FUNCTION_BLOCK FB_TaskMoveA_tilt EXTENDS FB_AbstructFuture
VAR_OUTPUT
END_VAR
VAR
	_v				: MC_LREAL;
	_a				: MC_LREAL;
	_d				: MC_LREAL;
	_j				: MC_LREAL;
	_dynamics		: DynamicConstraint_PathXY;
	_position 		: LREAL;
	_error_id		: UDINT;
	_fbMover		: POINTER TO MC_PlanarMover;
	_cmdFB			: MC_PlanarFeedback;
	_prohibit 		: BOOL;
	_abort_executor : FB_Executor;
	_state 			:UINT;
	_abort_state	:UINT;
END_VAR

{warning 'add method implementation '}
METHOD abort : BOOL
VAR_INST
	home_a :BOOL;
	home_b :BOOL;
END_VAR
_cmdFB.Update();
_state :=0;
CASE _abort_state OF
	0:
		IF _cmdFB.Active THEN
			_dynamics.SetValuesVADJ(2000,20000,200000,200000);
			home_a := FALSE;
			home_b := FALSE;
			//停止
			_fbMover^.Halt(_cmdFB,_dynamics);
			_abort_state := 1;
		ELSE
			abort := TRUE;
		END_IF
	1:
		IF _cmdFB.Done THEN
			IF _cmdFB.Error THEN
				abort := TRUE;
				_abort_state := 0;
				_error_id := _cmdFB.ErrorId;
			ELSE
				IF NOT home_a THEN
					_abort_state := 2;
				ELSIF NOT home_b THEN
					_abort_state := 3;
				ELSE
					abort := TRUE;
					_error_id := 0;
				END_IF
			END_IF
		END_IF
	2:
		_fbMover^.MoveA(_cmdFB,0,_dynamics);
		home_a := TRUE;
		_abort_state := 1;
	3:
		_fbMover^.MoveB(_cmdFB,0,_dynamics);
		home_b := TRUE;
		_abort_state := 1;
END_CASE
END_METHOD

{warning 'add method implementation '}
METHOD execute : BOOL
_cmdFB.Update();
_abort_state := 0;
CASE _state OF
	0:
		//直線運動
		IF NOT _cmdFB.Active AND NOT _cmdFB.Busy THEN
			_fbMover^.MoveA(_cmdFB,_position,_dynamics);
			_state := 1;
		END_IF
	1:
		//直線運動の完了フラグ待ち
		IF _cmdFB.Done THEN
			execute := TRUE;
			_error_id := 0;
		END_IF
		IF _cmdFB.Error THEN
			execute := TRUE;
			_error_id := _cmdFB.ErrorId;
		END_IF
END_CASE
END_METHOD

METHOD FB_init : BOOL
VAR_INPUT
	bInitRetains : BOOL; // if TRUE, the retain variables are initialized (warm start / cold start)
	bInCopyCode : BOOL;  // if TRUE, the instance afterwards gets moved into the copy code (online change)
	fbMover : REFERENCE TO MC_PlanarMover;
END_VAR
_fbMover := ADR(fbMover);
END_METHOD

{warning 'add method implementation '}
METHOD init : BOOL
IF _prohibit THEN
	_error_id := 16#80000000;
	init := TRUE;
ELSIF _v = 0 OR _a = 0 OR _d = 0 THEN
	_error_id := 1;
	init := TRUE;
ELSE
	_dynamics.SetValuesVADJ(_v, _a, _d, _j);
	_abort_executor.init();
	_error_id := 0;
	_state := 0;
	_abort_state := 0;
	init := TRUE;
END_IF
END_METHOD

{warning 'add property implementation'}
PROPERTY nErrorID : UDINT
GET
nErrorID := _error_id;
END_GET
END_PROPERTY

{warning 'add method implementation '}
METHOD quit : BOOL
init();
quit := TRUE;
END_METHOD

METHOD set_dynamics : BOOL
VAR_INPUT
	v: MC_LREAL;
	a: MC_LREAL;
	d: MC_LREAL;
	j: MC_LREAL;
END_VAR
_v := v;
_a := a;
_d := d;
_j := j;
set_dynamics := TRUE;
END_METHOD

METHOD set_target_position : BOOL
VAR_INPUT
	z: LREAL;
END_VAR
_position := z;

set_target_position := TRUE;
END_METHOD

END_FUNCTION_BLOCK

(* stored: Version 1.1.0.1, ProductVersion 3.1.4024.12
   POU FB_TaskMoveA_tilt: Id {fa3adf9d-2af0-4a8d-8b26-6e371a0f5aba}, SpecialFunc None
   Method abort: Id {eeecc789-f32f-4bf5-8281-de1db93e44bc}
   Method execute: Id {9b66e29d-a509-4db9-b77b-bcf9b0f95387}
   Method FB_init: Id {56269795-48db-41cc-b254-1e097d145e56}
   Method init: Id {157ada8f-e9dc-4d19-9683-6c15ed3e7958}
   Property nErrorID: Id {b2c64924-dcae-42c0-9c1d-7ccac65ca5de}
   Get Get: Id {e34175d1-be0a-4713-917f-72c5dcceacf0}
   Method quit: Id {812d5705-45b1-466a-9ae9-a82bec642401}
   Method set_dynamics: Id {97e6727e-9fa2-4ade-bdd1-fc9a068c1aa7}
   Method set_target_position: Id {c903e770-9c7a-4814-8d81-458589ee3655} *)
